TYPE T_ISO8601Time : STRING(30);
END_TYPE

(* stored: Version 1.1.0.1
   DUT T_ISO8601Time: Id {84fbd3a6-41be-4191-903a-48e8ae036a93} *)
